Staubli VAL3: prog.dtx

public string eventi
